FUNCTION_BLOCK AGRIPPER_MUX (* Composite FB wrapping other FBs *)
  (* Standard: 61499-2 *)
  (* Version 0.0, 2008-07-10, 4DIAC-IDE, 4DIAC-Consortium *)
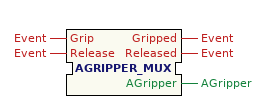
  EVENT_INPUT
    Grip; (* Confirmation from Plug *)
    Release; (* Indication from Plug *)
  END_EVENT
  EVENT_OUTPUT
    Gripped; (* Request from Socket *)
    Released; (* Response from Socket *)
  END_EVENT
  PLUGS
    AGripper : AGripper;
  END_PLUGS
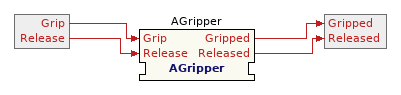
  EVENT_CONNECTIONS
    Grip TO AGripper.Grip;
    Release TO AGripper.Release;
    AGripper.Gripped TO Gripped;
    AGripper.Released TO Released;
  END_CONNECTIONS
END_FUNCTION_BLOCK
